FUNCTION_BLOCK FieldSignals_HMI (* Service Interface Function Block Type *)
  (* Standard: 61499-2 *)
  (* Version 0.0, 3/5/2026, Schneider Electric, template *)
  PACKAGE SE.Nereda;
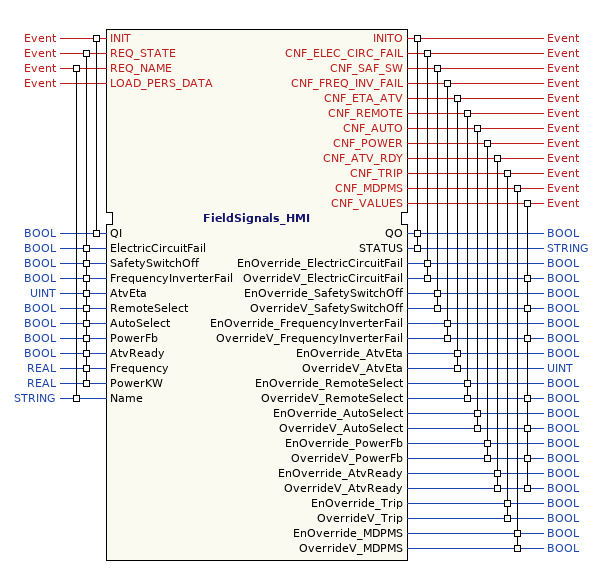
  EVENT_INPUT
    INIT WITH QI;
    REQ_STATE WITH ElectricCircuitFail, SafetySwitchOff, FrequencyInverterFail, AtvEta, RemoteSelect, AutoSelect, PowerFb, AtvReady, Frequency, PowerKW;
    REQ_NAME WITH Name;
    LOAD_PERS_DATA;
  END_EVENT
  EVENT_OUTPUT
    INITO WITH QO, STATUS;
    CNF_ELEC_CIRC_FAIL WITH OverrideV_ElectricCircuitFail, EnOverride_ElectricCircuitFail;
    CNF_SAF_SW WITH OverrideV_SafetySwitchOff, EnOverride_SafetySwitchOff;
    CNF_FREQ_INV_FAIL WITH OverrideV_FrequencyInverterFail, EnOverride_FrequencyInverterFail;
    CNF_ETA_ATV WITH OverrideV_AtvEta, EnOverride_AtvEta;
    CNF_REMOTE WITH OverrideV_RemoteSelect, EnOverride_RemoteSelect;
    CNF_AUTO WITH OverrideV_AutoSelect, EnOverride_AutoSelect;
    CNF_POWER WITH OverrideV_PowerFb, EnOverride_PowerFb;
    CNF_ATV_RDY WITH OverrideV_AtvReady, EnOverride_AtvReady;
    CNF_TRIP WITH EnOverride_Trip, OverrideV_Trip;
    CNF_MDPMS WITH EnOverride_MDPMS, OverrideV_MDPMS;
    CNF_VALUES WITH OverrideV_ElectricCircuitFail, OverrideV_SafetySwitchOff, OverrideV_FrequencyInverterFail, OverrideV_RemoteSelect, OverrideV_AutoSelect, OverrideV_PowerFb, OverrideV_AtvReady;
  END_EVENT
  VAR_INPUT
    QI : BOOL;
    ElectricCircuitFail : BOOL;
    SafetySwitchOff : BOOL;
    FrequencyInverterFail : BOOL;
    AtvEta : UINT;
    RemoteSelect : BOOL;
    AutoSelect : BOOL;
    PowerFb : BOOL;
    AtvReady : BOOL;
    Frequency : REAL;
    PowerKW : REAL;
    Name : STRING;
  END_VAR
  VAR_OUTPUT
    QO : BOOL; (* Event Output Qualifier *)
    STATUS : STRING; (* Service Status *)
    EnOverride_ElectricCircuitFail : BOOL;
    OverrideV_ElectricCircuitFail : BOOL;
    EnOverride_SafetySwitchOff : BOOL;
    OverrideV_SafetySwitchOff : BOOL;
    EnOverride_FrequencyInverterFail : BOOL;
    OverrideV_FrequencyInverterFail : BOOL;
    EnOverride_AtvEta : BOOL;
    OverrideV_AtvEta : UINT;
    EnOverride_RemoteSelect : BOOL;
    OverrideV_RemoteSelect : BOOL;
    EnOverride_AutoSelect : BOOL;
    OverrideV_AutoSelect : BOOL;
    EnOverride_PowerFb : BOOL;
    OverrideV_PowerFb : BOOL;
    EnOverride_AtvReady : BOOL;
    OverrideV_AtvReady : BOOL;
    EnOverride_Trip : BOOL;
    OverrideV_Trip : BOOL;
    EnOverride_MDPMS : BOOL;
    OverrideV_MDPMS : BOOL;
  END_VAR
  SERVICE /
    SEQUENCE 
    END_SEQUENCE
  END_SERVICE
END_FUNCTION_BLOCK
